{attribute 'GeneratedUsingTerminal: EK1100-0000-0018'}
{attribute addProperty BoxType "EK1100-0000-0018"}
{attribute addProperty Id "Beckhoff_EP3xxxEK1122Beckhoff_EP3xxxEK1122_039E50BA2708"}
{attribute addProperty CRC "2054902569"}
{attribute addProperty Size "2708"}
TYPE Beckhoff_EP3xxx_7A7B5329 EXTENDS EK1100_1FC0878B :
STRUCT
	{attribute addProperty Name "Beckhoff_EP3xxxEK1122"}
	{attribute addProperty PreviousPort "Beckhoff EP3xxx : B"}
	Beckhoff_EP3xxxEK1122 : Beckhoff_EP3xxxEK1122_039E50BA;
END_STRUCT
END_TYPE

(* stored: Version 1.2.0.0, ProductVersion 3.1.4024.9
   DUT Beckhoff_EP3xxx_7A7B5329: Id {8f4098c1-d6a1-4e91-9506-104454e35dcd} *)
